// TIA Portal V20 export
TYPE "UDT_SequenceInterface"
   STRUCT
      Error : Bool;
      Reset : Bool;
      SequenceReleased : Bool;
      SequenceRun : Bool;
      JobDone : Bool;
      StartRequest : Bool;
   END_STRUCT;
END_TYPE
